TYPE T_Dint : DINT; END_TYPE

(* stored: Version 1.1.0.1
   DUT T_Dint: Id {ac4c7b2c-812d-49cd-bad5-35d8cd449a8d} *)
